// positive edge detection
PROGRAM p05_posEdge
VAR
	S0: BOOL;
	M0: BOOL;
	M1: BOOL;
END_VAR

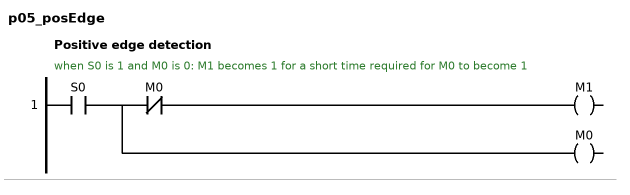
// NETWORK 1: Positive edge detection
// when S0 is 1 and M0 is 0: M1 becomes 1 for a short time required for M0 to become 1
M1 := S0 AND NOT M0;
M0 := S0;

END_PROGRAM

(* stored: Version 1.1.0.1, ProductVersion 3.1.4024.13
   POU p05_posEdge: Id {cc36aedf-cb5f-4fab-8107-5a25844d9856}, SpecialFunc None *)
